FUNCTION F_Temp_Write_Ramp_Value : BOOL
VAR_INPUT
	Module_Number	:WORD;
	Write_Value		:WORD;
END_VAR
VAR
END_VAR

F_Temp_Write_Ramp_Value:=F_Temp_Write_Value(Module_Number:=Module_Number,
											Command_Index:=161,
											Write_Value:=Write_Value);

END_FUNCTION

(* stored: Version 1.1.0.1
   POU F_Temp_Write_Ramp_Value: Id {255aca7b-5b9d-4bca-a5f5-a4d0271a5474}, SpecialFunc None *)
